Yaskawa INFORM job: SYS_FILTERS_START.JBI

/JOB
//NAME SYS_FILTERS_START
//POS
///NPOS 0,0,0,0,0,0
//INST
///DATE 2021/12/03 12:00
///ATTR SC,RW
///GROUP1 RB1
NOP
DOUT OT#(20) OFF
DOUT OT#(21) OFF
WAIT T=1.00
DOUT OT#(20) ON
WAIT T=7.00
DOUT OT#(21) ON
END
